TYPE T_Ctrl_SIf_BCC_Out :
STRUCT
END_STRUCT
END_TYPE

(* stored: Version 1.1.0.1, ProductVersion 3.1.0.19
   DUT T_Ctrl_SIf_BCC_Out: Id {26bec251-a379-496c-8912-16bc1106a856} *)
